(* Logix 5000 project; controller PLC2_Project_6_Hourmeter Emulate 5570 rev 20.11; software revision 20.00 *)
// Plant hourmeter with a reset button

TASK MainTask (continuous, watchdog 500 ms) : MainProgram

MODULES
   Local : Emulate 5570 (ICP 1, rev 20.11)
END_MODULES

PROGRAM MainProgram   (* main routine MainRoutine *)
VAR
   Button_HourMeterReset : BOOL; {access Read Only}
   Hourmeter_HundredsHours : DINT; {access Read Only}
   Hourmeter_Minutes : DINT; {access Read Only}
   Hourmeter_Seconds : DINT; {access Read Only}
   Hourmeter_ThousandsHours : DINT; {access Read Only}
   I_0_0 : BOOL; {access Read Only}   // Fake input
   I_0_1 : BOOL; {access Read Only}   // Fake input
   ONS_HourmeterReset : BOOL; {access Read Only}
   SecondsTimer : TIMER := (PRE := 1000); {access Read Only}
   StartCounting : BOOL; {access Read Only}
   System_Running : BOOL; {access Read Only}   // Is the plant running?
END_VAR

ROUTINE Hourmeter   (* ladder *)
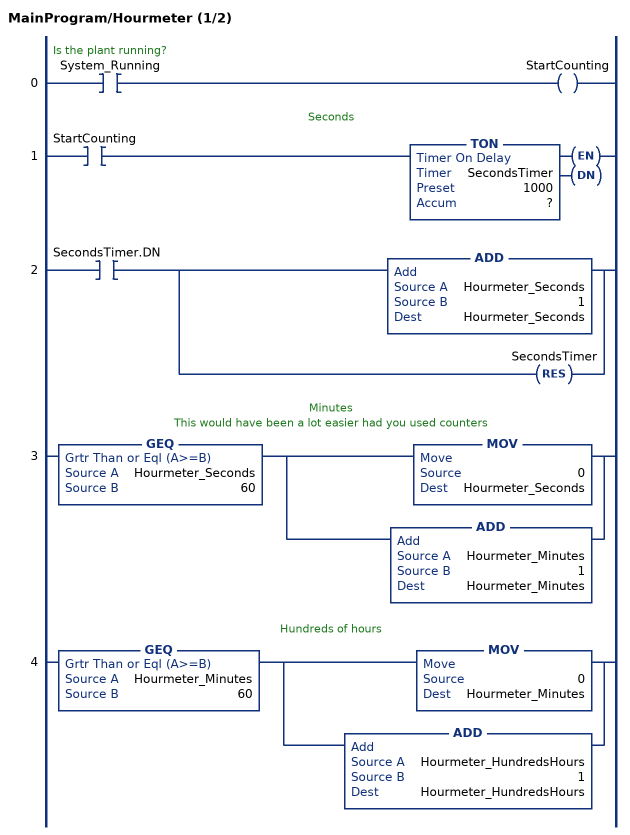
   0: XIC(System_Running)OTE(StartCounting);
   // Seconds
   1: XIC(StartCounting)TON(SecondsTimer,?,?);
   2: XIC(SecondsTimer.DN)[ADD(Hourmeter_Seconds,1,Hourmeter_Seconds) ,RES(SecondsTimer) ];
   // Minutes
   // This would have been a lot easier had you used counters
   3: GEQ(Hourmeter_Seconds,60)[MOV(0,Hourmeter_Seconds) ,ADD(Hourmeter_Minutes,1,Hourmeter_Minutes) ];
   // Hundreds of hours
   4: GEQ(Hourmeter_Minutes,60)[MOV(0,Hourmeter_Minutes) ,ADD(Hourmeter_HundredsHours,1,Hourmeter_HundredsHours) ];
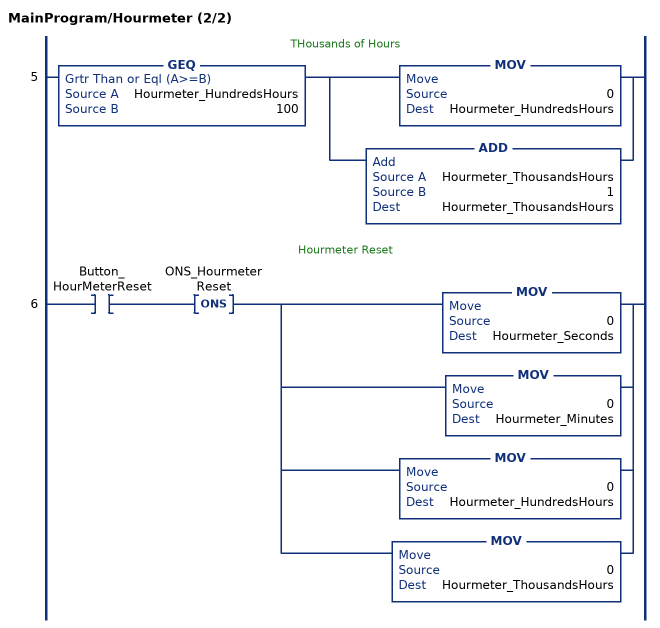
   // THousands of Hours
   5: GEQ(Hourmeter_HundredsHours,100)[MOV(0,Hourmeter_HundredsHours) ,ADD(Hourmeter_ThousandsHours,1,Hourmeter_ThousandsHours) ];
   // Hourmeter Reset
   6: XIC(Button_HourMeterReset)ONS(ONS_HourmeterReset)[MOV(0,Hourmeter_Seconds) ,MOV(0,Hourmeter_Minutes) ,MOV(0,Hourmeter_HundredsHours) ,MOV(0,Hourmeter_ThousandsHours) ];
END_ROUTINE

ROUTINE InputOutput   (* ladder *)
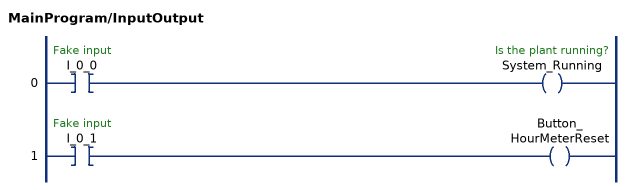
   0: XIC(I_0_0)OTE(System_Running);
   1: XIC(I_0_1)OTE(Button_HourMeterReset);
END_ROUTINE

ROUTINE MainRoutine   (* ladder *)
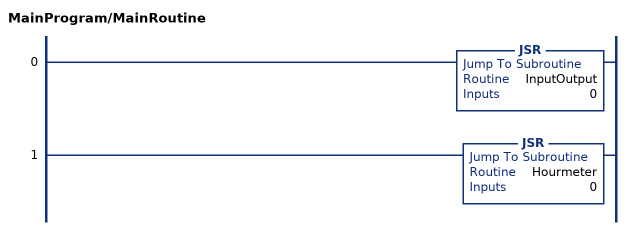
   0: JSR(InputOutput,0);
   1: JSR(Hourmeter,0);
END_ROUTINE
END_PROGRAM
